// Mitsubishi GX Works2 project: BookEX6_36 DataTable   PLC: Q13UDV

// global labels: Global
VAR_GLOBAL
  bVar0 AT M5000 : BOOL;
  abArray0 AT M5010 : ARRAY [0..49] OF BOOL;
  sStr0 AT D5000 : STRING[199];
  sStr1 AT D5100 : STRING[199];
  sStr2 AT D5200 : STRING[199];
  sStr3 AT D5300 : STRING[199];
  sStr4 AT D5400 : STRING[199];
  sStr5 AT D5500 : STRING[199];
  sStr6 AT D5600 : STRING[199];
  sStr7 AT D5700 : STRING[199];
  sStr8 AT D5800 : STRING[199];
  sStr9 AT D5900 : STRING[199];
  iVar0 AT D4500 : INT;
  iVar1 AT D4501 : INT;
  iVar2 AT D4502 : INT;
  iVar3 AT D4503 : INT;
  iVar4 AT D4504 : INT;
  iVar5 AT D4505 : INT;
  iVar6 AT D4506 : INT;
  iVar7 AT D4507 : INT;
  iVar8 AT D4508 : INT;
  iVar9 AT D4509 : INT;
  dVar0 AT D4510 : DINT;
  dVar1 AT D4512 : DINT;
  dVar2 AT D4514 : DINT;
  dVar3 AT D4516 : DINT;
  dVar4 AT D4518 : DINT;
  dVar5 AT D4520 : DINT;
  dVar6 AT D4522 : DINT;
  dVar7 AT D4524 : DINT;
  dVar8 AT D4526 : DINT;
  dVar9 AT D4528 : DINT;
  wVar0 AT D4530 : WORD;
  wVar1 AT D4531 : WORD;
  wVar2 AT D4532 : WORD;
  wVar3 AT D4533 : WORD;
  wVar4 AT D4534 : WORD;
  wVar5 AT D4535 : WORD;
  wVar6 AT D4536 : WORD;
  wVar7 AT D4537 : WORD;
  wVar8 AT D4538 : WORD;
  wVar9 AT D4539 : WORD;
  dwVar0 AT D4540 : DWORD;
  dwVar1 AT D4542 : DWORD;
  dwVar2 AT D4544 : DWORD;
  dwVar3 AT D4546 : DWORD;
  dwVar4 AT D4548 : DWORD;
  dwVar5 AT D4550 : DWORD;
  dwVar6 AT D4552 : DWORD;
  dwVar7 AT D4554 : DWORD;
  dwVar8 AT D4556 : DWORD;
  dwVar9 AT D4558 : DWORD;
  fsVar0 AT D4560 : REAL;
  fsVar1 AT D4562 : REAL;
  fsVar2 AT D4564 : REAL;
  fsVar3 AT D4566 : REAL;
  fsVar4 AT D4568 : REAL;
  fsVar5 AT D4570 : REAL;
  fsVar6 AT D4572 : REAL;
  fsVar7 AT D4574 : REAL;
  fsVar8 AT D4576 : REAL;
  fsVar9 AT D4578 : REAL;
  fdVar0 AT D4580 : LREAL;
  tTime0 AT D4620 : TIME;
  tTime1 AT D4622 : TIME;
  tTime2 AT D4624 : TIME;
  tTime3 AT D4626 : TIME;
  tTime4 AT D4628 : TIME;
  tTime5 AT D4630 : TIME;
  tTime6 AT D4632 : TIME;
  tTime7 AT D4634 : TIME;
  tTime8 AT D4636 : TIME;
  tTime9 AT D4638 : TIME;
  tTime10 AT D4640 : TIME;
  bVar1 AT M5001 : BOOL;
  bVar2 AT M5002 : BOOL;
  bVar3 AT M5003 : BOOL;
  bVar4 AT M5004 : BOOL;
  bVar5 AT M5005 : BOOL;
  bVar6 AT M5006 : BOOL;
  bVar7 AT M5007 : BOOL;
  bVar8 AT M5008 : BOOL;
  bVar9 AT M5009 : BOOL;
  abArray1 AT M5060 : ARRAY [0..49] OF BOOL;
  abArray2 AT M5110 : ARRAY [0..49] OF BOOL;
  abArray3 AT M5160 : ARRAY [0..49] OF BOOL;
  abArray4 AT M5210 : ARRAY [0..49] OF BOOL;
  abArray5 AT M5260 : ARRAY [0..49] OF BOOL;
  abArray6 AT M5310 : ARRAY [0..49] OF BOOL;
  abArray7 AT M5360 : ARRAY [0..49] OF BOOL;
  abArray8 AT M5410 : ARRAY [0..49] OF BOOL;
  abArray9 AT M5460 : ARRAY [0..49] OF BOOL;
  fdVar1 AT D4584 : LREAL;
  fdVar2 AT D4588 : LREAL;
  fdVar3 AT D4592 : LREAL;
  fdVar4 AT D4596 : LREAL;
  fdVar5 AT D4600 : LREAL;
  fdVar6 AT D4604 : LREAL;
  fdVar7 AT D4608 : LREAL;
  fdVar8 AT D4612 : LREAL;
  fdVar9 AT D4616 : LREAL;
  afsPen0 AT D2000 : ARRAY [0..499] OF REAL;
  afsPen1 AT D3000 : ARRAY [0..499] OF REAL;
  adwD10 AT D10 : ARRAY [0..9] OF DWORD;
  awD10 AT D10 : ARRAY [0..19] OF WORD;
  aiD100 AT D100 : ARRAY [0..9] OF INT;
  aiD110 AT D110 : ARRAY [0..9] OF INT;
  aiD120 AT D120 : ARRAY [0..9] OF INT;
  aiD130 AT D130 : ARRAY [0..9] OF INT;
  abM10 AT M10 : ARRAY [0..19] OF BOOL;
  gaiIndex AT D4700 : ARRAY [0..255] OF INT;
  gaiFIFO AT D4800 : ARRAY [0..255] OF INT;
END_VAR
// user libraries (not included): HMI

FUNCTION_BLOCK FIFO8
VAR_INPUT
  i_Din : INT;
  b_R : BOOL;
  b_W : BOOL;
  b_Reset : BOOL;
END_VAR
VAR_OUTPUT
  i_Dout : INT;
  b_Empty : BOOL;
  b_Full : BOOL;
END_VAR
VAR
  aiBuff : ARRAY [0..7] OF INT;
  iGet : INT;
  iPut : INT;
END_VAR
VAR_OUTPUT
  i_Buff1 : INT;
  i_Buff2 : INT;
  i_Buff3 : INT;
  i_Buff4 : INT;
  i_Buff5 : INT;
  i_Buff6 : INT;
  i_Buff7 : INT;
  i_Buff8 : INT;
  i_Get : INT;
  i_Put : INT;
END_VAR
VAR
  iTmp : INT;
END_VAR
VAR_INPUT
  b_EN : BOOL;
END_VAR
;
IF b_Reset THEN
	iGet := 0;
	iPut := 0;
	b_Full := FALSE;
	b_Empty := TRUE;
	FOR iTmp := 0 TO 7 DO 
		aiBuff[iTmp] := 0;
	END_FOR;
	i_Dout := 0;
ELSE
	IF NOT b_Empty AND b_R AND b_EN THEN
		i_Dout := aiBuff[iGet];
		IF iGet >= 7 THEN
			iGet := 0;
		ELSE
			iGet := iGet+1;
		END_IF;
		b_Empty := iGet = iPut;
		b_Full := FALSE;
	END_IF;
	IF NOT b_Full AND b_W AND b_EN THEN
		aiBuff[iPut] := i_Din;
		IF iPut >= 7 THEN
			iPut := 0;
		ELSE
			iPut := iPut+1;
		END_IF;
		b_Full := iPut = iGet;
		b_Empty := FALSE;
	END_IF;
END_IF;

i_Buff1 := aiBuff[0];
i_Buff2 := aiBuff[1];
i_Buff3 := aiBuff[2];
i_Buff4 := aiBuff[3];
i_Buff5 := aiBuff[4];
i_Buff6 := aiBuff[5];
i_Buff7 := aiBuff[6];
i_Buff8 := aiBuff[7];
i_Get := iGet;
i_Put := iPut;
END_FUNCTION_BLOCK

FUNCTION_BLOCK MultiFIFO
VAR_INPUT
  b_GetCnt : BOOL;
  b_Get1st : BOOL;
  b_Get2nd : BOOL;
  b_AddWait : BOOL;
  b_DelWait : BOOL;
  b_InsWait : BOOL;
  i_BlkNo : INT;
  i_InData : INT;
END_VAR
VAR_OUTPUT
  i_Cnt : INT;
  i_OtData : INT;
END_VAR
VAR
  ix : INT;
  iy : INT;
  iz : INT;
  aiIndex : ARRAY [0..255] OF INT;
END_VAR
VAR_OUTPUT
  ai_CpIndex : ARRAY [0..255] OF INT;
  ai_CpFIFO : ARRAY [0..255] OF INT;
END_VAR
VAR
  aiFIFO : ARRAY [0..255] OF INT;
END_VAR
VAR_INPUT
  b_Reset : BOOL;
END_VAR
VAR
  ii : INT;
END_VAR
;
IF LDP(TRUE, b_Reset) THEN
	FOR ix := 0 TO 255 DO 
		aiIndex[ix] := 0;
		aiFIFO[ix] := 0;
	END_FOR;
END_IF;

IF LDP(TRUE, b_GetCnt) THEN
	i_Cnt := aiIndex[i_BlkNo] - aiIndex[i_BlkNo-1];
END_IF;

IF LDP(TRUE, b_Get1st) THEN
	ix := aiIndex[i_BlkNo] - aiIndex[i_BlkNo-1];
	IF ix = 0 THEN
		i_Cnt := 0;
		i_OtData := 0;
	ELSE
		i_Cnt := ix;
		i_OtData := aiFIFO[aiIndex[i_BlkNo-1]];
	END_IF;
END_IF;

IF LDP(TRUE, b_Get2nd) THEN
	ix := aiIndex[i_BlkNo] - aiIndex[i_BlkNo-1];
	IF ix < 2 THEN
		i_Cnt := 0;
		i_OtData := 0;
	ELSE
		i_Cnt := ix;
		i_OtData := aiFIFO[aiIndex[i_BlkNo-1]+1];
	END_IF;
END_IF;

IF LDP(TRUE, b_AddWait) AND i_BlkNo <> 0 AND i_InData <> 0 THEN
	iy := i_InData;
	ii := aiIndex[i_BlkNo];
	FOR ix := ii TO 255 DO 
		iz := aiFIFO[ix];
		aiFIFO[ix] := iy;
		iy := iz;
	END_FOR;
	FOR ix := i_BlkNo TO 255 DO 
		aiIndex[ix] := aiIndex[ix] + 1;
	END_FOR;	
	i_Cnt := aiIndex[i_BlkNo] - aiIndex[i_BlkNo-1];
	i_OtData := aiFIFO[aiIndex[i_BlkNo-1]];
END_IF;

IF LDP(TRUE, b_DelWait) AND i_BlkNo <> 0 AND i_InData <> 0 THEN
	iz := aiIndex[i_BlkNo] - aiIndex[i_BlkNo-1];
	IF iz <> 0 THEN
			iy := aiIndex[i_BlkNo-1];
			FOR ii := iy TO 255 DO 
				aiFIFO[ii] := aiFIFO[ii+1];
			END_FOR;
			FOR ii := i_BlkNo TO 255 DO 	
				aiIndex[ii] := aiIndex[ii] - 1;
			END_FOR;
	END_IF;
	i_Cnt := aiIndex[i_BlkNo] - aiIndex[i_BlkNo-1];
	i_OtData := aiFIFO[aiIndex[i_BlkNo-1]];
END_IF;

IF LDP(TRUE, b_InsWait) AND i_BlkNo <> 0 AND i_InData <> 0 THEN
	iy := i_InData;
	ii := aiIndex[i_BlkNo-1];
	FOR ix := ii TO 255 DO 
		iz := aiFIFO[ix];
		aiFIFO[ix] := iy;
		iy := iz;
	END_FOR;
	FOR ix := i_BlkNo TO 255 DO 
		aiIndex[ix] := aiIndex[ix] + 1;
	END_FOR;
	i_Cnt := aiIndex[i_BlkNo] - aiIndex[i_BlkNo-1];
	i_OtData := aiFIFO[aiIndex[i_BlkNo-1]];
END_IF;

ai_CpIndex := aiIndex;
ai_CpFIFO := aiFIFO;
END_FUNCTION_BLOCK

FUNCTION_BLOCK STACK8
VAR_INPUT
  i_Din : INT;
  b_R : BOOL;
  b_W : BOOL;
  b_Reset : BOOL;
END_VAR
VAR_OUTPUT
  i_Dout : INT;
  b_Empty : BOOL;
  b_Full : BOOL;
END_VAR
VAR
  aiBuff : ARRAY [0..7] OF INT;
  iPtr : INT;
END_VAR
VAR_OUTPUT
  i_Buff1 : INT;
  i_Buff2 : INT;
  i_Buff3 : INT;
  i_Buff4 : INT;
  i_Buff5 : INT;
  i_Buff6 : INT;
  i_Buff7 : INT;
  i_Buff8 : INT;
  i_Ptr : INT;
END_VAR
VAR_INPUT
  b_EN : BOOL;
END_VAR
VAR
  ix : INT;
END_VAR
;
IF b_Reset THEN
	iPtr := 0;
	b_Full := FALSE;
	b_Empty := TRUE;
	FOR ix := 0 TO 7 DO 
		aiBuff[ix] := 0;
	END_FOR;
	i_Dout := 0;
ELSE
	IF NOT b_Empty AND  b_R AND b_EN THEN
		iPtr := iPtr - 1;
		i_Dout := aiBuff[iPtr];
		b_Empty := iPtr = 0;
		b_Full := FALSE;
	END_IF;
	IF NOT b_Full AND b_W AND b_EN THEN
		aiBuff[iPtr] := i_Din;
		iPtr := iPtr + 1;
		b_Full := iPtr > 7;
		b_Empty := FALSE;
	END_IF;
END_IF;
i_Buff1 := aiBuff[0];
i_Buff2 := aiBuff[1];
i_Buff3 := aiBuff[2];
i_Buff4 := aiBuff[3];
i_Buff5 := aiBuff[4];
i_Buff6 := aiBuff[5];
i_Buff7 := aiBuff[6];
i_Buff8 := aiBuff[7];
i_Ptr := iPtr;
END_FUNCTION_BLOCK

PROGRAM ExDataTable
(* structured ladder/FBD written out as ST: instructions are called as NAME(EN, inputs, outputs); _pN, _eN, _tN stand for wires *)
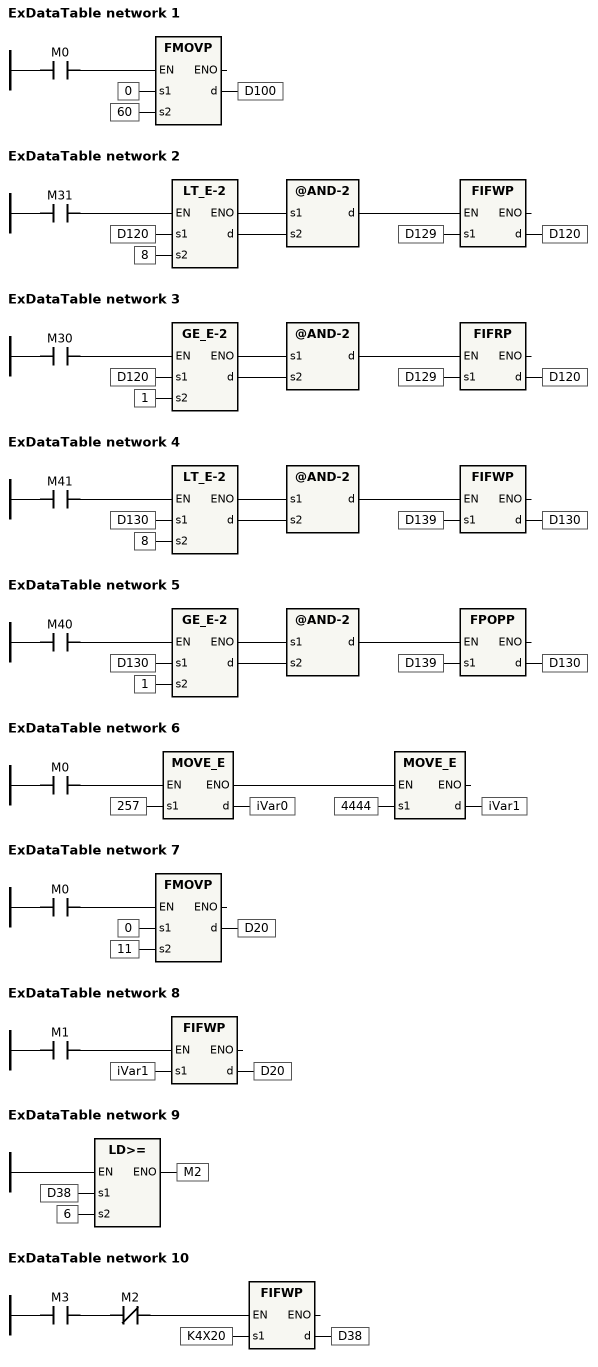
(* network 1 *)
FMOVP(M0, 0, 60, D100);
(* network 2 *)
_e2 := LT_E(M31, D120, 8, _t1);
FIFWP(@AND-2(_e2, _t1), D129, D120);
(* network 3 *)
_e2 := GE_E(M30, D120, 1, _t1);
FIFRP(@AND-2(_e2, _t1), D129, D120);
(* network 4 *)
_e2 := LT_E(M41, D130, 8, _t1);
FIFWP(@AND-2(_e2, _t1), D139, D130);
(* network 5 *)
_e2 := GE_E(M40, D130, 1, _t1);
FPOPP(@AND-2(_e2, _t1), D139, D130);
(* network 6 *)
_e1 := MOVE_E(M0, 257, iVar0);
MOVE_E(_e1, 4444, iVar1);
(* network 7 *)
FMOVP(M0, 0, 11, D20);
(* network 8 *)
FIFWP(M1, iVar1, D20);
(* network 9 *)
_e1 := LD>=(TRUE, D38, 6);
M2 := _e1;
(* network 10 *)
FIFWP(M3 AND NOT M2, K4X20, D38);
END_PROGRAM

PROGRAM ExFIFO8
VAR
  FIFO8_1 : FIFO8;
  STACK8_1 : STACK8;
END_VAR
(* structured ladder/FBD written out as ST: instructions are called as NAME(EN, inputs, outputs); _pN, _eN, _tN stand for wires *)
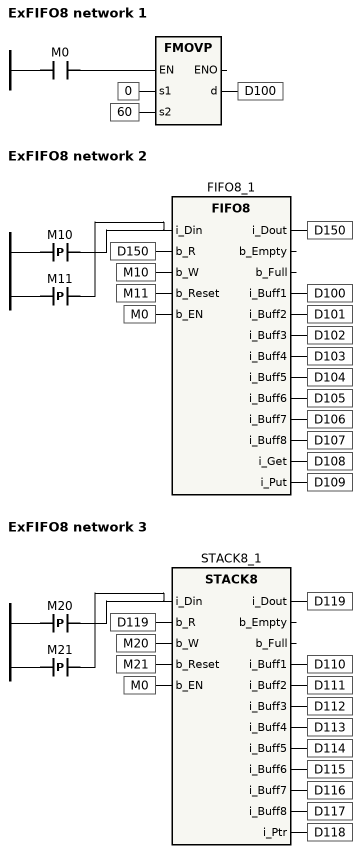
(* network 1 *)
FMOVP(M0, 0, 60, D100);
(* network 2 *)
FIFO8_1(i_Din := LDP(TRUE, M10) OR LDP(TRUE, M11), b_R := D150, b_W := M10, b_Reset := M11, b_EN := M0, i_Dout => D150, i_Buff1 => D100, i_Buff2 => D101, i_Buff3 => D102, i_Buff4 => D103, i_Buff5 => D104, i_Buff6 => D105, i_Buff7 => D106, i_Buff8 => D107, i_Get => D108, i_Put => D109);
(* network 3 *)
STACK8_1(i_Din := LDP(TRUE, M20) OR LDP(TRUE, M21), b_R := D119, b_W := M20, b_Reset := M21, b_EN := M0, i_Dout => D119, i_Buff1 => D110, i_Buff2 => D111, i_Buff3 => D112, i_Buff4 => D113, i_Buff5 => D114, i_Buff6 => D115, i_Buff7 => D116, i_Buff8 => D117, i_Ptr => D118);
END_PROGRAM

PROGRAM ExMultiFIFO
VAR
  MultiFIFO_1 : MultiFIFO;
END_VAR
(* structured ladder/FBD written out as ST: instructions are called as NAME(EN, inputs, outputs); _pN, _eN, _tN stand for wires *)
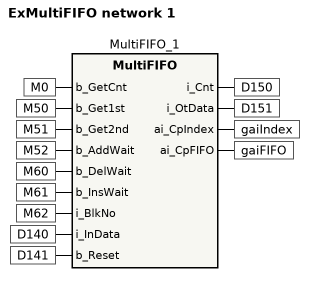
(* network 1 *)
MultiFIFO_1(b_GetCnt := M0, b_Get1st := M50, b_Get2nd := M51, b_AddWait := M52, b_DelWait := M60, b_InsWait := M61, i_BlkNo := M62, i_InData := D140, b_Reset := D141, i_Cnt => D150, i_OtData => D151, ai_CpIndex => gaiIndex, ai_CpFIFO => gaiFIFO);
END_PROGRAM

PROGRAM ExFIFR
(* structured ladder/FBD written out as ST: instructions are called as NAME(EN, inputs, outputs); _pN, _eN, _tN stand for wires *)
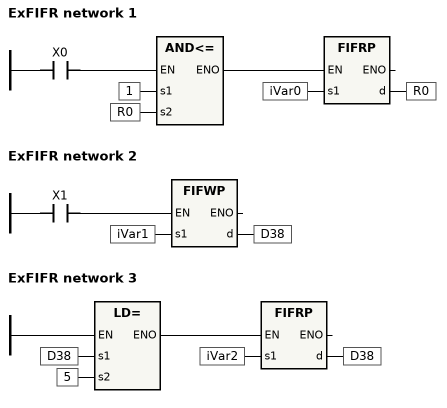
(* network 1 *)
_e1 := AND<=(X0, 1, R0);
FIFRP(_e1, iVar0, R0);
(* network 2 *)
FIFWP(X1, iVar1, D38);
(* network 3 *)
_e1 := LD=(TRUE, D38, 5);
FIFRP(_e1, iVar2, D38);
END_PROGRAM

PROGRAM ExFPOP
(* structured ladder/FBD written out as ST: instructions are called as NAME(EN, inputs, outputs); _pN, _eN, _tN stand for wires *)
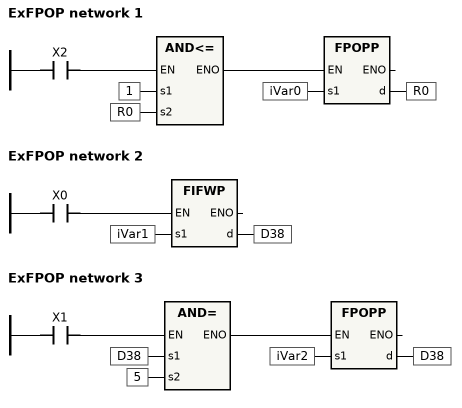
(* network 1 *)
_e1 := AND<=(X2, 1, R0);
FPOPP(_e1, iVar0, R0);
(* network 2 *)
FIFWP(X0, iVar1, D38);
(* network 3 *)
_e1 := AND=(X1, D38, 5);
FPOPP(_e1, iVar2, D38);
END_PROGRAM

PROGRAM ExFDEL
(* structured ladder/FBD written out as ST: instructions are called as NAME(EN, inputs, outputs); _pN, _eN, _tN stand for wires *)
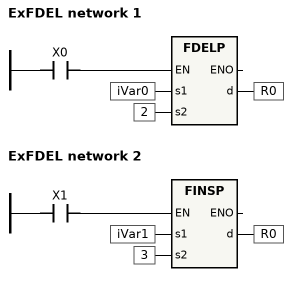
(* network 1 *)
FDELP(X0, iVar0, 2, R0);
(* network 2 *)
FINSP(X1, iVar1, 3, R0);
END_PROGRAM
